/// Change configuration of selected user frame number
FUNCTION_BLOCK WriteFrameDataFB EXTENDS RobotLibraryBaseFB
// ------------------------------------------------------------------------- 
//  SRCI Robot Library                                                
// ------------------------------------------------------------------------- 
//                                                                           
//  Object:      WriteFrameDataFB                                       
//  Author:      Thorsten Brach                                                
//  Date:        2024-06-01
//
//  Description:                                              
//   
//                                                                           
//  Copyright: 
//    (C) 2024 Thorsten Brach. All rights reserved                                                                         
//                                                                           
//  Disclaimer:                                                                           
//    This project is provided without any guarantee and can be used for   
//    private and commercial purposes. Any commercial use is at the user’s 
//    own risk and responsibility.
//
// -------------------------------------------------------------------------
VAR_INPUT 
  /// Start of the command at the rising edge
  Execute            : BOOL;
  /// Processing Mode
  ProcessingMode     : ProcessingMode;
  /// Frame index M
  /// • 0: WCS (default) O
  /// • 1..254: UCS (User frames)
  FrameNo            : USINT;
  /// Frame data (see chapter 5.5.6.2)
  FrameData          : FrameData;
  /// Defines the target sequence in which the command will be executed
  SequenceFlag       : SequenceFlag;
END_VAR
VAR_OUTPUT
  /// The command has been completed successfully
  Done               : BOOL;
  /// FB is being processed
  Busy               : BOOL;
  /// Command is transferred and confirmed by the RC
  CommandBuffered    : BOOL;
  /// The command was aborted by another command
  CommandAborted     : BOOL;
  /// TRUE, while command is interrupted during execution and can be continued.
  CommandInterrupted : BOOL;
END_VAR

                  
                

METHOD PROTECTED OnCall
VAR_IN_OUT
  /// Robot assignment of function
  AxesGroup         : AxesGroup; 
END_VAR
                        
                      
END_METHOD
END_FUNCTION_BLOCK

/// Write integer values on RC
FUNCTION_BLOCK WriteIntegersFB EXTENDS RobotLibraryBaseFB
// ------------------------------------------------------------------------- 
//  SRCI Robot Library                                                
// ------------------------------------------------------------------------- 
//                                                                           
//  Object:      WriteIntegersFB                                       
//  Author:      Thorsten Brach                                                
//  Date:        2024-06-01
//
//  Description:                                              
//   
//                                                                           
//  Copyright: 
//    (C) 2024 Thorsten Brach. All rights reserved                                                                         
//                                                                           
//  Disclaimer:                                                                           
//    This project is provided without any guarantee and can be used for   
//    private and commercial purposes. Any commercial use is at the user’s 
//    own risk and responsibility.
//
// -------------------------------------------------------------------------
VAR_INPUT
  /// Start of the command at the rising edge
  Execute            : BOOL;
  /// Processing Mode
  ProcessingMode     : ProcessingMode;
  /// Specifies the desired target values that shall be written
  Index              : ARRAY[0..6] OF USINT; 
  /// Array value of integers
  Values             : ARRAY[0..6] OF INT;
  /// Set TRUE to prioritize the execution of this command in the defined target sequence.
  HighPriority       : BOOL;
  /// Defines the target sequence in which the command will be executed
  SequenceFlag       : SequenceFlag;
  /// ID of associated trigger function:
  /// •  0: No Trigger (default)  No trigger related behavior
  /// • >0: Trigger - Start executing when the trigger function with the identical EmitterID is triggered.
  /// Always positive.
  /// For more information, see chapter 5.5.12 Triggers
  ListenerID         : SINT;
END_VAR
VAR_OUTPUT
  /// The command has been completed successfully
  Done               : BOOL;
  /// FB is being processed
  Busy               : BOOL;
  /// Command is transferred and confirmed by the RC
  CommandBuffered    : BOOL;
  /// The command was aborted by another command.
  CommandAborted     : BOOL;
  /// TRUE, while command is interrupted during execution and can be continued
  CommandInterrupted : BOOL;
  /// Receiving of input parameter values has been acknowledged by RC
  ParameterAccepted  : BOOL;
  /// Unique system-generated ID of the "Action" when the function is triggered.
  /// • >0: The "Action" is started by the trigger function with identical FollowID.
  /// • <0: The "Action" is stopped by the trigger function with identical FollowID.
  /// For more information see chapter 5.5.12.4.
  OriginID           : USINT;
  /// Relates to ListenerID >0 
  /// Number of successful trigger -based command invocations
  /// For more information refer to chapter 5.5.12.4.
  InvocationCounter  : USINT;
END_VAR

                  
                

METHOD PROTECTED OnCall
VAR_IN_OUT
  /// Robot assignment of function
  AxesGroup         : AxesGroup; 
END_VAR
                        
                      
END_METHOD
END_FUNCTION_BLOCK

/// Change configuration of selected payload number
FUNCTION_BLOCK WriteLoadDataFB EXTENDS RobotLibraryBaseFB
// ------------------------------------------------------------------------- 
//  SRCI Robot Library                                                
// ------------------------------------------------------------------------- 
//                                                                           
//  Object:      WriteLoadDataFB                                       
//  Author:      Thorsten Brach                                                
//  Date:        2024-06-01
//
//  Description:                                              
//   
//                                                                           
//  Copyright: 
//    (C) 2024 Thorsten Brach. All rights reserved                                                                         
//                                                                           
//  Disclaimer:                                                                           
//    This project is provided without any guarantee and can be used for   
//    private and commercial purposes. Any commercial use is at the user’s 
//    own risk and responsibility.
//
// -------------------------------------------------------------------------
VAR_INPUT
  /// Start of the command at the rising edge
  Execute            : BOOL;
  /// Processing Mode
  ProcessingMode     : ProcessingMode;
  /// Load index
  /// •      0: (default) - Not possible to write
  /// • 1..254: Load data
  LoadNo             : USINT;
  /// Load data (see chapter 5.5.6.4)
  LoadData           : LoadData;
  /// Defines the target sequence in which the command will be executed
  SequenceFlag       : SequenceFlag;
END_VAR
VAR_OUTPUT
  /// The command has been completed successfully
  Done               : BOOL;
  /// FB is being processed
  Busy               : BOOL;
  /// Command is transferred and confirmed by the RC
  CommandBuffered    : BOOL;
  /// The command was aborted by another command
  CommandAborted     : BOOL;
  /// TRUE, while command is interrupted during execution and can be continued.
  CommandInterrupted : BOOL;
END_VAR

                  
                

METHOD PROTECTED OnCall
VAR_IN_OUT
  /// Robot assignment of function
  AxesGroup         : AxesGroup; 
END_VAR
                        
                      
END_METHOD
END_FUNCTION_BLOCK

/// Write real values on RC
FUNCTION_BLOCK WriteRealsFB EXTENDS RobotLibraryBaseFB
// ------------------------------------------------------------------------- 
//  SRCI Robot Library                                                
// ------------------------------------------------------------------------- 
//                                                                           
//  Object:      WriteRealsFB                                       
//  Author:      Thorsten Brach                                                
//  Date:        2024-06-01
//
//  Description:                                              
//   
//                                                                           
//  Copyright: 
//    (C) 2024 Thorsten Brach. All rights reserved                                                                         
//                                                                           
//  Disclaimer:                                                                           
//    This project is provided without any guarantee and can be used for   
//    private and commercial purposes. Any commercial use is at the user’s 
//    own risk and responsibility.
//
// -------------------------------------------------------------------------
VAR_INPUT
  /// Start of the command at the rising edge
  Execute            : BOOL;
  /// Processing Mode
  ProcessingMode     : ProcessingMode;
  /// Specifies the desired target values that shall be written
  Index              : ARRAY[0..6] OF USINT; 
  /// Array value of reas
  Values             : ARRAY[0..6] OF REAL;
  /// Set TRUE to prioritize the execution of this command in the defined target sequence.
  HighPriority       : BOOL;
  /// Defines the target sequence in which the command will be executed
  SequenceFlag       : SequenceFlag;
  /// ID of associated trigger function:
  /// •  0: No Trigger (default)  No trigger related behavior
  /// • >0: Trigger - Start executing when the trigger function with the identical EmitterID is triggered.
  /// Always positive.
  /// For more information, see chapter 5.5.12 Triggers
  ListenerID         : SINT;
END_VAR
VAR_OUTPUT
  /// The command has been completed successfully
  Done               : BOOL;
  /// FB is being processed
  Busy               : BOOL;
  /// Command is transferred and confirmed by the RC
  CommandBuffered    : BOOL;
  /// The command was aborted by another command.
  CommandAborted     : BOOL;
  /// TRUE, while command is interrupted during execution and can be continued
  CommandInterrupted : BOOL;
  /// Receiving of input parameter values has been acknowledged by RC
  ParameterAccepted  : BOOL;
  /// Unique system-generated ID of the "Action" when the function is triggered.
  /// • >0: The "Action" is started by the trigger function with identical FollowID.
  /// • <0: The "Action" is stopped by the trigger function with identical FollowID.
  /// For more information see chapter 5.5.12.4.
  OriginID           : USINT;
  /// Relates to ListenerID >0 
  /// Number of successful trigger -based command invocations
  /// For more information refer to chapter 5.5.12.4.
  InvocationCounter  : USINT;
END_VAR

                  
                

METHOD PROTECTED OnCall
VAR_IN_OUT
  /// Robot assignment of function
  AxesGroup         : AxesGroup; 
END_VAR
                        
                      
END_METHOD
END_FUNCTION_BLOCK

/// Write default values of dynamic parameters used by move commands
FUNCTION_BLOCK WriteRobotDefaultDynamicsFB EXTENDS RobotLibraryBaseFB
// ------------------------------------------------------------------------- 
//  SRCI Robot Library                                                
// ------------------------------------------------------------------------- 
//                                                                           
//  Object:      WriteRobotDefaultDynamicsFB                                       
//  Author:      Thorsten Brach                                                
//  Date:        2024-06-01
//
//  Description:                                              
//   
//                                                                           
//  Copyright: 
//    (C) 2024 Thorsten Brach. All rights reserved                                                                         
//                                                                           
//  Disclaimer:                                                                           
//    This project is provided without any guarantee and can be used for   
//    private and commercial purposes. Any commercial use is at the user’s 
//    own risk and responsibility.
//
// -------------------------------------------------------------------------
VAR_INPUT
  /// Start of the command at the rising edge
  Execute                : BOOL;
  /// Processing Mode
  ProcessingMode         : ProcessingMode;
  /// Default dynamics values according to Table 6-141.
  DynamicValues          : DefaultDynamics;
END_VAR
VAR_OUTPUT
  /// The command has been completed successfully
  Done                   : BOOL;
  /// FB is being processed
  Busy                   : BOOL;
  /// Command is transferred and confirmed by the RC
  CommandBuffered        : BOOL;
  /// The command was aborted by another command
  CommandAborted         : BOOL;
  /// TRUE, while command is interrupted during execution and can be continued.
  CommandInterrupted     : BOOL;
  /// Commanded dynamics values according to Table 6-141.
  DefaultDynamicValues   : DefaultDynamics;
END_VAR

                  
                

METHOD PROTECTED OnCall
VAR_IN_OUT
  /// Robot assignment of function
  AxesGroup         : AxesGroup; 
END_VAR
                        
                      
END_METHOD
END_FUNCTION_BLOCK

/// Write reference values of robot dynamics for path movement
FUNCTION_BLOCK WriteRobotReferenceDynamicsFB EXTENDS RobotLibraryBaseFB
// ------------------------------------------------------------------------- 
//  SRCI Robot Library                                                
// ------------------------------------------------------------------------- 
//                                                                           
//  Object:      WriteRobotReferenceDynamicsFB                                       
//  Author:      Thorsten Brach                                                
//  Date:        2024-06-01
//
//  Description:                                              
//   
//                                                                           
//  Copyright: 
//    (C) 2024 Thorsten Brach. All rights reserved                                                                         
//                                                                           
//  Disclaimer:                                                                           
//    This project is provided without any guarantee and can be used for   
//    private and commercial purposes. Any commercial use is at the user’s 
//    own risk and responsibility.
//
// -------------------------------------------------------------------------
VAR_INPUT
  /// Start of the command at the rising edge
  Execute                : BOOL;
  /// Processing Mode
  ProcessingMode         : ProcessingMode;
  /// Reference dynamics values according TO Table 6-134.
  DynamicValues          : ReferenceDynamics;
END_VAR
VAR_OUTPUT
  /// The command has been completed successfully
  Done                   : BOOL;
  /// FB is being processed
  Busy                   : BOOL;
  /// Command is transferred and confirmed by the RC
  CommandBuffered        : BOOL;
  /// The command was aborted by another command
  CommandAborted         : BOOL;
  /// TRUE, while command is interrupted during execution and can be continued.
  CommandInterrupted     : BOOL;
  /// Commanded reference dynamics values according to Table 6-134
  ReferenceDynamicValues : ReferenceDynamics;
END_VAR

                  
                

METHOD PROTECTED OnCall
VAR_IN_OUT
  /// Robot assignment of function
  AxesGroup         : AxesGroup; 
END_VAR
                        
                      
END_METHOD
END_FUNCTION_BLOCK

/// Change robot limits of robot axes (degree)
FUNCTION_BLOCK WriteRobotSWLimitsFB EXTENDS RobotLibraryBaseFB
// ------------------------------------------------------------------------- 
//  SRCI Robot Library                                                
// ------------------------------------------------------------------------- 
//                                                                           
//  Object:      WriteRobotSWLimitsFB                                       
//  Author:      Thorsten Brach                                                
//  Date:        2024-06-01
//
//  Description:                                              
//   
//                                                                           
//  Copyright: 
//    (C) 2024 Thorsten Brach. All rights reserved                                                                         
//                                                                           
//  Disclaimer:                                                                           
//    This project is provided without any guarantee and can be used for   
//    private and commercial purposes. Any commercial use is at the user’s 
//    own risk and responsibility.
//
// -------------------------------------------------------------------------
VAR_INPUT
  /// Start of the command at the rising edge
  Execute                : BOOL;
  /// Limits for joints and external axes according to Table 6-180.
  LimitValues            : SWLimits;
  /// Reset limits to RC specific factory settings
  ResetToFactoryDefaults : BOOL;;
END_VAR
VAR_OUTPUT
  /// The command has been completed successfully
  Done                   : BOOL;
  /// FB is being processed
  Busy                   : BOOL;
  /// Command is transferred and confirmed by the RC
  CommandBuffered        : BOOL;
  /// TRUE, when Software limits were overwritten but not activated on RC until a restart of the RC
  RestartRequested       : BOOL;
END_VAR

                  
                

METHOD PROTECTED OnCall
VAR_IN_OUT
  /// Robot assignment of function
  AxesGroup         : AxesGroup; 
END_VAR
                        
                      
END_METHOD
END_FUNCTION_BLOCK

/// Write specific parameter of the robot
FUNCTION_BLOCK WriteSystemVariableFB EXTENDS RobotLibraryBaseFB
// ------------------------------------------------------------------------- 
//  SRCI Robot Library                                                
// ------------------------------------------------------------------------- 
//                                                                           
//  Object:      WriteSystemVariableFB                                       
//  Author:      Thorsten Brach                                                
//  Date:        2024-06-01
//
//  Description:                                              
//   
//                                                                           
//  Copyright: 
//    (C) 2024 Thorsten Brach. All rights reserved                                                                         
//                                                                           
//  Disclaimer:                                                                           
//    This project is provided without any guarantee and can be used for   
//    private and commercial purposes. Any commercial use is at the user’s 
//    own risk and responsibility.
//
// -------------------------------------------------------------------------
VAR_INPUT
  /// Start of the command at the rising edge
  Execute            : BOOL;
  /// Processing Mode
  ProcessingMode     : ProcessingMode;
  /// Defines the parameter list which should be used:
  /// • FALSE: Standardized parameter list (default):
  ///          -  Read parameters on the RC based on a standardized parameter list
  /// • TRUE: Manufacturer specific parameter list:
  ///        -  Read parameters on the RC based on robot manufacturers-specific parameter lists
  RCParameter        : BOOL;
  /// Requested parameter ID in selected parameter list.
  /// •          0: undefined (default)
  /// • 1..65 535: Parameter ID
  ParameterID        : ARRAY[0..7] OF UINT;
  /// ID of the requested sub parameter in selected parameter list.
  /// • 0: ID 0 (default) (relates only to parameters without sub parameters)
  /// • 1..255: Indices 1 to 255 (relates only to parameters with sub parameters)
  SubParameterID     : ARRAY[0..7] OF USINT;  
  /// Parameter data type as specified in Table 6-621.
  DataType           : ARRAY[0..7] OF USINT;
  /// Parameter data addressed by input values of ParameterID[0] and SubParameterID[0]
  Data_0             : ARRAY[0..3] OF BYTE;
  /// Parameter data addressed by input values of ParameterID[1] and SubParameterID[1]
  Data_1             : ARRAY[0..3] OF BYTE;
  /// Parameter data addressed by input values of ParameterID[2] and SubParameterID[2]
  Data_2             : ARRAY[0..3] OF BYTE;
  /// Parameter data addressed by input values of ParameterID[3] and SubParameterID[3]
  Data_3             : ARRAY[0..3] OF BYTE;
  /// Parameter data addressed by input values of ParameterID[4] and SubParameterID[4]
  Data_4             : ARRAY[0..3] OF BYTE;
  /// Parameter data addressed by input values of ParameterID[5] and SubParameterID[5]
  Data_5             : ARRAY[0..3] OF BYTE;
  /// Parameter data addressed by input values of ParameterID[6] and SubParameterID[6]
  Data_6             : ARRAY[0..3] OF BYTE;
  /// Parameter data addressed by input values of ParameterID[7] and SubParameterID[7]
  Data_7             : ARRAY[0..3] OF BYTE;
  /// Defines the target sequence in which the command will be executed
  SequenceFlag       : SequenceFlag;
  /// ID of associated trigger function:
  /// •  0: No Trigger (default)  No trigger related behavior
  /// • >0: Trigger - Start executing when the trigger function with the identical EmitterID is triggered.
  /// Always positive.
  /// For more information, see chapter 5.5.12 Triggers
  ListenerID         : SINT;
END_VAR
VAR_OUTPUT
  /// The command has been completed successfully
  Done               : BOOL;
  /// FB is being processed
  Busy               : BOOL;
  /// Command is transferred and confirmed by the RC
  CommandBuffered    : BOOL;
  /// The command was aborted by another command.
  CommandAborted     : BOOL;
  /// TRUE, while command is interrupted during execution and can be continued
  CommandInterrupted : BOOL;
  /// TRUE, when parameters were overwritten but not activated on RC until a restart of the RC
  RestartRequested   : BOOL;
  /// Unique system-generated ID of the "Action" when the function is triggered.
  /// • >0: The "Action" is started by the trigger function with identical FollowID.
  /// • <0: The "Action" is stopped by the trigger function with identical FollowID.
  /// For more information see chapter 5.5.12.4 EmitterID, ListenerID, FollowID and OriginID
  OriginID           : INT;
  /// Relates to ListenerID >0
  /// Number of successful trigger -based command invocations
  /// For more information refer to chapter 5.5.12.4.
  InvocationCounter  : USINT;
END_VAR

                  
                

METHOD PROTECTED OnCall
VAR_IN_OUT
  /// Robot assignment of function
  AxesGroup         : AxesGroup; 
END_VAR
                        
                      
END_METHOD
END_FUNCTION_BLOCK

/// Change configuration of selected tool number
FUNCTION_BLOCK WriteToolDataFB EXTENDS RobotLibraryBaseFB
// ------------------------------------------------------------------------- 
//  SRCI Robot Library                                                
// ------------------------------------------------------------------------- 
//                                                                           
//  Object:      WriteToolDataFB                                       
//  Author:      Thorsten Brach                                                
//  Date:        2024-06-01
//
//  Description:                                              
//   
//                                                                           
//  Copyright: 
//    (C) 2024 Thorsten Brach. All rights reserved                                                                         
//                                                                           
//  Disclaimer:                                                                           
//    This project is provided without any guarantee and can be used for   
//    private and commercial purposes. Any commercial use is at the user’s 
//    own risk and responsibility.
//
// -------------------------------------------------------------------------
VAR_INPUT
  /// Start of the command at the rising edge
  Execute            : BOOL;
  /// Processing Mode
  ProcessingMode     : ProcessingMode;
  /// Tool index
  /// •      0: Flange (default) Not possible to change
  /// • 1..254: Tool Frame
  ToolNo            : USINT;
  /// Tool data (see chapter 5.5.6.3)
  ToolData          : ToolData;
  /// Defines the target sequence in which the command will be executed
  SequenceFlag       : SequenceFlag;
END_VAR
VAR_OUTPUT
  /// The command has been completed successfully
  Done               : BOOL;
  /// FB is being processed
  Busy               : BOOL;
  /// Command is transferred and confirmed by the RC
  CommandBuffered    : BOOL;
  /// The command was aborted by another command
  CommandAborted     : BOOL;
  /// TRUE, while command is interrupted during execution and can be continued.
  CommandInterrupted : BOOL;
END_VAR

                  
                

METHOD PROTECTED OnCall
VAR_IN_OUT
  /// Robot assignment of function
  AxesGroup         : AxesGroup; 
END_VAR
                        
                      
END_METHOD
END_FUNCTION_BLOCK

/// Define work area
FUNCTION_BLOCK WriteWorkAreaFB EXTENDS RobotLibraryBaseFB
// ------------------------------------------------------------------------- 
//  SRCI Robot Library                                                
// ------------------------------------------------------------------------- 
//                                                                           
//  Object:      WriteWorkAreaFB                                       
//  Author:      Thorsten Brach                                                
//  Date:        2024-06-01
//
//  Description:                                              
//   
//                                                                           
//  Copyright: 
//    (C) 2024 Thorsten Brach. All rights reserved                                                                         
//                                                                           
//  Disclaimer:                                                                           
//    This project is provided without any guarantee and can be used for   
//    private and commercial purposes. Any commercial use is at the user’s 
//    own risk and responsibility.
//
// -------------------------------------------------------------------------
VAR_INPUT
  /// Start of the command at the rising edge
  Execute            : BOOL;
  /// Processing Mode
  ProcessingMode     : ProcessingMode;
  /// Index of the robot work area
  /// • 0 (default)..254
  WorkAreaNo         : USINT;
  /// Data specific to the work area requested by Index.
  WorkAreaData       : RobotWorkArea;
END_VAR
VAR_OUTPUT
  /// The command has been completed successfully
  Done               : BOOL;
  /// FB is being processed
  Busy               : BOOL;
  /// Command is transferred and confirmed by the RC
  CommandBuffered    : BOOL;
END_VAR

                  
                

METHOD PROTECTED OnCall
VAR_IN_OUT
  /// Robot assignment of function
  AxesGroup         : AxesGroup; 
END_VAR
                        
                      
END_METHOD
END_FUNCTION_BLOCK

FUNCTION_BLOCK ActiveCommandRegisterFB
// ------------------------------------------------------------------------- 
//  SRCI Robot Library                                                
// ------------------------------------------------------------------------- 
//                                                                           
//  Object:      ActiveCommandRegisterFB                                       
//  Author:      Thorsten Brach                                                
//  Date:        2024-06-01
//
//  Description:                                              
//   
//                                                                           
//  Copyright: 
//    (C) 2024 Thorsten Brach. All rights reserved                                                                         
//                                                                           
//  Disclaimer:                                                                           
//    This project is provided without any guarantee and can be used for   
//    private and commercial purposes. Any commercial use is at the user’s 
//    own risk and responsibility.
//
// -------------------------------------------------------------------------
VAR_INPUT
  /// Active Command Register
  Register            : ARRAY [1..RobotLibraryParameter.ACTIVE_CMD_REGISTER_ENTRIES_MAX] OF AxesGroupAcyclicAcrEntry;
END_VAR

VAR_OUTPUT
  /// Size of the register 
  Size                : UINT := DINT_TO_UINT(RobotLibraryParameter.ACTIVE_CMD_REGISTER_ENTRIES_MAX);
  /// Execution Order List 
  ExecutionOrderList  : AxesGroupAcyclicExecutionOrderList;
END_VAR

VAR
  /// last used unique ID 
  LastUniqueID        : UDINT;
END_VAR

                  OnCall();


                

METHOD INTERNAL AddCmd : UDINT
VAR_INPUT
  /// Reference to the corresponding command-FB to enable a callback mechanism
  rCommandFB   : REFERENCE TO RobotLibraryBaseFB;
END_VAR

VAR
  /// internal index for loops
 _idx : DINT;
END_VAR
                        FOR _idx := 1 TO RobotLibraryParameter.ACTIVE_CMD_REGISTER_ENTRIES_MAX
DO
  IF ( Register[_idx].State = ActiveCommandRegisterState.IS_FREE )
  THEN
    Register[_idx].State                        := ActiveCommandRegisterState.IS_PROCESSING;
    Register[_idx].UniqueID                     := CreateUniqueID();
    Register[_idx].rCommandFB                   := rCommandFB;

    // check reference to command FB
    IF (__ISVALIDREF(Register[_idx].rCommandFB))
    THEN
      Register[_idx].Command[1].Payload    := rCommandFB.CommandData.Payload;
      Register[_idx].Command[1].PayloadLen := rCommandFB.CommandData.PayloadLen;
      Register[_idx].Command[1].PayLoadPtr := 0;
      Register[_idx].Command[1].State      := BufferStateCmd.CREATED;
		END_IF
  
    // return Unique ID
    AddCmd := Register[_idx].UniqueID;
    EXIT;
	END_IF
END_FOR
                      
END_METHOD

METHOD INTERNAL CreateUniqueID : UDINT
VAR_INPUT
END_VAR
                        // inc last unique ID 
LastUniqueID := LastUniqueID + 1;
// return unique ID
CreateUniqueID := LastUniqueID;
                      
END_METHOD

METHOD INTERNAL OnCall
                        
                      
END_METHOD

METHOD OnlineChange : DINT
VAR_INPUT
  /// unique ID 
  UniqueID     : UDINT;
  /// Reference to the corresponding command-FB to enable a callback mechanism
  rCommandFB   : REFERENCE TO RobotLibraryBaseFB;
END_VAR

VAR
  /// internal index for loops
 _idx : DINT;
END_VAR
                        OnlineChange := -1;

// Check command FB reference is valid ?
IF ( NOT __ISVALIDREF(rCommandFB))
THEN
  RETURN;
END_IF

FOR _idx := 1 TO RobotLibraryParameter.ACTIVE_CMD_REGISTER_ENTRIES_MAX
DO
  // check unique ID found ?
  IF ( Register[_idx].UniqueID = UniqueID ) 
  THEN  
    // update reference to command FB
    Register[_idx].rCommandFB := rCommandFB;
    // Return result OK
    OnlineChange := RobotLibraryConstants.OK;
    EXIT;
  END_IF
END_FOR
                      
END_METHOD

METHOD RemoveCmd
VAR_INPUT
 /// unique ID
 UniqueID : UDINT;  
END_VAR

VAR
  /// internal index
 _idx : DINT;
END_VAR
                        FOR _idx := 1 TO RobotLibraryParameter.ACTIVE_CMD_REGISTER_ENTRIES_MAX
DO
  // check unique ID found and not yet sended ?
  IF (( Register[_idx].UniqueID         = UniqueID               ) AND
      ( Register[_idx].Command[1].State < BufferStateCmd.SENDING ))       
  THEN  
    // delete register entry
    MemSet(ADR(Register[_idx]), 0 , SIZEOF(Register[_idx]));
    EXIT;
  END_IF
END_FOR
                      
END_METHOD

METHOD SortList : ARRAY [1..RobotLibraryParameter.ACTIVE_CMD_REGISTER_ENTRIES_MAX] OF UINT;
VAR_INPUT
  List : ARRAY [1..RobotLibraryParameter.ACTIVE_CMD_REGISTER_ENTRIES_MAX] OF UINT;
END_VAR

VAR
  i   : DINT;
  j   : DINT;
  tmp : UINT;
END_VAR
                        // Bubble Sort 
FOR i := 1 TO RobotLibraryParameter.ACTIVE_CMD_REGISTER_ENTRIES_MAX
DO
  FOR j := 1 TO RobotLibraryParameter.ACTIVE_CMD_REGISTER_ENTRIES_MAX - 1
  DO
    IF ( List[j] > List[j+1])
    THEN
       Tmp := List[j];         
       List[j]   := List[j+1];
       List[j+1] := Tmp;
    END_IF
  END_FOR 
END_FOR

// return sorted list
SortList := List;
                      
END_METHOD

METHOD UpdateExecutionOrderList
VAR
  _idxReg  : DINT;
  _idxList : DINT := 1;
END_VAR
                        FOR _idxReg := 1 TO RobotLibraryParameter.ACTIVE_CMD_REGISTER_ENTRIES_MAX
DO
  IF (( Register[_idxReg].State              = ActiveCommandRegisterState.IS_PROCESSING ) AND
      ( Register[_idxReg].Response[1].State  =             BufferStateRsp.EMPTY         ))     
  THEN
    ;
  END_IF
END_FOR
                      
END_METHOD
END_FUNCTION_BLOCK

{attribute 'pack_mode' := '1'} 
FUNCTION_BLOCK RecvData
// ------------------------------------------------------------------------- 
//  SRCI Robot Library                                                
// ------------------------------------------------------------------------- 
//                                                                           
//  Object:      RecvData                                       
//  Author:      Thorsten Brach                                                
//  Date:        2024-06-01
//
//  Description:                                              
//   
//                                                                           
//  Copyright: 
//    (C) 2024 Thorsten Brach. All rights reserved                                                                         
//                                                                           
//  Disclaimer:                                                                           
//    This project is provided without any guarantee and can be used for   
//    private and commercial purposes. Any commercial use is at the user’s 
//    own risk and responsibility.
//
// -------------------------------------------------------------------------
VAR_INPUT
  /// Payload
  Payload    : ARRAY [0..RobotLibraryParameter.TELEGRAM_PAYLOAD_MAX] OF BYTE;
  /// Payload length
  PayloadLen : UDINT;
  /// Payload pointer
  PayloadPtr : DINT;
END_VAR

                  
                

/// returns a ArmConfigParameter from the payload buffer from the current payload pointer address and increase the payload pointer afterwards
METHOD GetArmConfig : ArmConfigParameter
VAR
  /// temporary byte
 _tmpByte : BYTE;
END_VAR
                        // get 1st Byte
_tmpByte := GetByte();

GetArmConfig.Shoulder.0 := _tmpByte.0;
GetArmConfig.Elbow.0    := _tmpByte.1;
GetArmConfig.Wrist.0    := _tmpByte.2;

// get 2nd byte to inc the PayloadPointer
_tmpByte := GetByte();
                      
END_METHOD

/// returns a BOOL from the payload buffer from the current payload pointer address and increase the payload pointer afterwards
METHOD GetBool : BOOL
                        // copy data
GetBool := Payload[PayloadPtr].0;
// inc payload pointer 
PayloadPtr := PayloadPtr + SIZEOF(BYTE);
                      
END_METHOD

/// returns a BYTE from the payload buffer from the current payload pointer address and increase the payload pointer afterwards
METHOD GetByte : BYTE
                        // copy data
GetByte := Payload[PayloadPtr];
// inc payload pointer 
PayloadPtr := PayloadPtr + SIZEOF(BYTE);
                      
END_METHOD

/// returns a DWORD from the payload buffer from the current payload pointer address and increase the payload pointer afterwards
METHOD GetDword : DWORD
                        // copy data
MemCpy(ADR(GetDword), ADR(Payload[PayloadPtr]), SIZEOF(DWORD));
// inc payload pointer 
PayloadPtr := PayloadPtr + SIZEOF(DWORD);
                      
END_METHOD

/// returns the 1st halfe BYTE from the payload buffer from the current payload pointer address and increase the payload pointer afterwards
METHOD GetHalfeByte1 : BYTE
VAR_INPUT
  /// Increase payload pointer 
  IncPayloadPtr : BOOL;
END_VAR

VAR
  /// temporary byte
 _tmpByte : BYTE;
END_VAR
                        // copy data
_tmpByte := Payload[PayloadPtr];

GetHalfeByte1.0 := _tmpByte.0;
GetHalfeByte1.1 := _tmpByte.1;
GetHalfeByte1.2 := _tmpByte.2;
GetHalfeByte1.3 := _tmpByte.3;


IF (IncPayloadPtr)
THEN  
  // inc payload pointer
  PayloadPtr := PayloadPtr + SIZEOF(BYTE);
END_IF

                      
END_METHOD

/// returns the 1st halfe BYTE from the payload buffer from the current payload pointer address and increase the payload pointer afterwards
METHOD GetHalfeByte2 : BYTE
VAR_INPUT
  /// Increase payload pointer 
  IncPayloadPtr : BOOL;
END_VAR

VAR
  /// temporary byte
 _tmpByte : BYTE;
END_VAR
                        // copy data
_tmpByte := Payload[PayloadPtr];

GetHalfeByte2.0 := _tmpByte.4;
GetHalfeByte2.1 := _tmpByte.5;
GetHalfeByte2.2 := _tmpByte.6;
GetHalfeByte2.3 := _tmpByte.7;

IF (IncPayloadPtr)
THEN  
  // inc payload pointer
  PayloadPtr := PayloadPtr + SIZEOF(BYTE);
END_IF

                      
END_METHOD

/// returns a INT from the payload buffer from the current payload pointer address and increase the payload pointer afterwards
METHOD GetInt : INT
                        // copy data
MemCpy(ADR(GetInt), ADR(Payload[PayloadPtr]), SIZEOF(INT));
// swap byte order
GetInt := SwapInt(GetInt);
// inc payload pointer   
PayloadPtr := PayloadPtr + SIZEOF(INT);
                      
END_METHOD

/// returns a REAL from the payload buffer from the current payload pointer address and increase the payload pointer afterwards
METHOD GetReal : REAL
                        // copy data
MemCpy(ADR(GetReal), ADR(Payload[PayloadPtr]), SIZEOF(REAL));
// swap byte order
GetReal := SwapReal(GetReal);
// inc payload pointer   
PayloadPtr := PayloadPtr + SIZEOF(Real);
                      
END_METHOD

/// returns a SINT from the payload buffer from the current payload pointer address and increase the payload pointer afterwards
METHOD GetSint : SINT
                        // copy data
MemCpy(ADR(GetSint), ADR(Payload[PayloadPtr]), SIZEOF(SINT));
// inc payload pointer 
PayloadPtr := PayloadPtr + SIZEOF(SINT);
                      
END_METHOD

/// returns a TurnNumber from the payload buffer from the current payload pointer address and increase the payload pointer afterwards
METHOD GetTurnNumbers : TurnNumber
                        GetTurnNumbers.J1Turns := BYTE_TO_SINT(GetHalfeByte1(FALSE));
GetTurnNumbers.J2Turns := BYTE_TO_SINT(GetHalfeByte2(TRUE));

GetTurnNumbers.J3Turns := BYTE_TO_SINT(GetHalfeByte1(FALSE));
GetTurnNumbers.J4Turns := BYTE_TO_SINT(GetHalfeByte2(TRUE));

GetTurnNumbers.J5Turns := BYTE_TO_SINT(GetHalfeByte1(FALSE));
GetTurnNumbers.J6Turns := BYTE_TO_SINT(GetHalfeByte2(TRUE));

GetTurnNumbers.E1Turns := BYTE_TO_SINT(GetByte());
                      
END_METHOD

/// returns a UINT from the payload buffer from the current payload pointer address and increase the payload pointer afterwards
METHOD GetUint : UINT
                        // copy data
MemCpy(ADR(GetUint), ADR(Payload[PayloadPtr]), SIZEOF(UINT));
// swap byte order
GetUint := SwapUint(GetUint);
// inc payload pointer   
PayloadPtr := PayloadPtr + SIZEOF(UINT);
                      
END_METHOD

/// returns a USINT from the payload buffer from the current payload pointer address and increase the payload pointer afterwards
METHOD GetUsint : USINT
                        // copy data
MemCpy(ADR(GetUsint), ADR(Payload[PayloadPtr]), SIZEOF(USINT));
// inc payload pointer 
PayloadPtr := PayloadPtr + SIZEOF(USINT);
                      
END_METHOD

/// returns a WORD from the payload buffer from the current payload pointer address and increase the payload pointer afterwards
METHOD GetWord : WORD
                        // copy data
MemCpy(ADR(GetWord), ADR(Payload[PayloadPtr]), SIZEOF(WORD));
// swap byte order
GetWord := SwapWord(GetWord);
// inc payload pointer   
PayloadPtr := PayloadPtr + SIZEOF(WORD);
                      
END_METHOD

/// Resets the payload pointer to start address
METHOD ResetPointer
VAR_INPUT
END_VAR
                        // Reset payload pointer
PayloadPtr := 0;
                      
END_METHOD

/// returns a FragmentAction from the payload buffer from the current payload pointer address and increase the payload pointer afterwards
METHOD GetFragmentAction : FragmentAction
VAR
  /// temporary byte
 _tmpByte : BYTE;
END_VAR
                        // copy data
_tmpByte := Payload[PayloadPtr];

GetFragmentAction.Complete := _tmpByte.0;
GetFragmentAction.Reset    := _tmpByte.1;
GetFragmentAction.Clear    := _tmpByte.2;
GetFragmentAction.BIT03    := _tmpByte.3;
GetFragmentAction.BIT04    := _tmpByte.4;
GetFragmentAction.BIT05    := _tmpByte.5;
GetFragmentAction.BIT06    := _tmpByte.6;
GetFragmentAction.BIT07    := _tmpByte.7;

// inc payload pointer   
PayloadPtr := PayloadPtr + SIZEOF(BYTE);
                      
END_METHOD
END_FUNCTION_BLOCK

{attribute 'pack_mode' := '1'} 
FUNCTION_BLOCK SendData
// ------------------------------------------------------------------------- 
//  SRCI Robot Library                                                
// ------------------------------------------------------------------------- 
//                                                                           
//  Object:      SendData                                      
//  Author:      Thorsten Brach                                                
//  Date:        2024-06-01
//
//  Description:                                              
//    
//                                                                           
//  Copyright: 
//    (C) 2024 Thorsten Brach. All rights reserved                                                                         
//                                                                           
//  Disclaimer:                                                                           
//    This project is provided without any guarantee and can be used for   
//    private and commercial purposes. Any commercial use is at the user’s 
//    own risk and responsibility.
//
// -------------------------------------------------------------------------
VAR_INPUT
  /// Payload
  Payload    : ARRAY [0..RobotLibraryParameter.TELEGRAM_PAYLOAD_MAX] OF BYTE;
  /// Payload length
  PayloadLen : UDINT;
  /// Payload pointer
  PayloadPtr : UDINT;
END_VAR

                  
                

/// Adds a BOOL to the payload buffer, increase the payload pointer and returns the payload lenght
METHOD AddBool : UDINT
VAR_INPUT
  /// Value to add
  Value : BOOL;
END_VAR

VAR
  /// temporary byte
 _tmpByte : BYTE := 0;
END_VAR
                        _tmpByte.0 := Value;
// copy data 
MemCpy( ADR(Payload[PayloadPtr]), ADR(_tmpByte), SIZEOF(_tmpByte));
// inc payload pointer 
PayloadPtr := PayloadPtr + SIZEOF(_tmpByte);
// return payload len
AddBool := PayloadLen := PayloadPtr;
                      
END_METHOD

/// Adds a BYTE to the payload buffer, increase the payload pointer and returns the payload lenght
METHOD AddByte : UDINT
VAR_INPUT
  /// Value to add
  Value : BYTE;
END_VAR
                        Value := Value;
// copy data 
MemCpy( ADR(Payload[PayloadPtr]), ADR(Value), SIZEOF(Value));
// inc payload pointer 
PayloadPtr := PayloadPtr + SIZEOF(Value);
// return payload len
AddByte := PayloadLen := PayloadPtr;
                      
END_METHOD

/// Adds a DataBlock to the payload buffer, increase the payload pointer and returns the payload lenght
METHOD AddDataBlock : UDINT
VAR_INPUT
  /// Value to add
  pValue : POINTER TO BYTE;
  /// Size of data block
  Size   : UDINT;
END_VAR
                        IF (pValue = 0) OR (Size = 0 )
THEN
  RETURN;
END_IF

// copy data 
MemCpy( ADR(Payload[PayloadPtr]), pValue, Size);
// inc payload pointer 
PayloadPtr := PayloadPtr + Size;
// return payload len
AddDataBlock := PayloadLen := PayloadPtr;
                      
END_METHOD

/// Adds two halfe BYTE to the payload buffer , increase the payload pointer and returns the payload lenght
METHOD AddHalfBytes : UDINT
VAR_INPUT
  /// Value to add
  Value1 : BYTE;
  /// Value to add
  Value2 : BYTE;
END_VAR

VAR
  /// internal value
 _value : BYTE;
END_VAR
                        _value := CombineHalfBytes(Value1,Value2);
// copy data 
MemCpy( ADR(Payload[PayloadPtr]), ADR(_value), SIZEOF(_value));
// inc payload pointer 
PayloadPtr := PayloadPtr + SIZEOF(_value);
// return payload len
AddHalfBytes := PayloadLen := PayloadPtr;
                      
END_METHOD

/// Adds a REAL to the payload buffer , increase the payload pointer and returns the payload lenght
METHOD AddReal : UDINT
VAR_INPUT
  /// Value to add
  Value : REAL;
END_VAR
                        // swap byte order
Value := SwapReal(Value);
// copy data 
MemCpy( ADR(Payload[PayloadPtr]), ADR(Value), SIZEOF(Value));
// inc data index 
PayloadPtr := PayloadPtr + SIZEOF(Value);
// return payload len
AddReal := PayloadLen := PayloadPtr;
                      
END_METHOD

/// Adds a SINT to the payload buffer, increase the payload pointer and returns the payload lenght
METHOD AddSint : UDINT
VAR_INPUT
  /// Value to add
  Value : SINT;
END_VAR
                        Value := Value;
// copy data 
MemCpy( ADR(Payload[PayloadPtr]), ADR(Value), SIZEOF(Value));
// inc payload pointer 
PayloadPtr := PayloadPtr + SIZEOF(Value);
// return payload len
AddSint := PayloadLen := PayloadPtr;
                      
END_METHOD

/// Adds a TIME to the payload buffer , increase the payload pointer and returns the payload lenght
METHOD AddTime : UDINT
VAR_INPUT
  /// Value to add
  Value : TOD;
END_VAR
                        // swap byte order
Value := SwapTime(Value);
// copy data 
MemCpy( ADR(Payload[PayloadPtr]), ADR(Value), SIZEOF(Value));
// inc data index 
PayloadPtr := PayloadPtr + SIZEOF(Value);
// return payload len
AddTime := PayloadLen := PayloadPtr;
                      
END_METHOD

/// Adds a UINT to the payload buffer , increase the payload pointer and returns the payload lenght
METHOD AddUint : UDINT
VAR_INPUT
  /// Value to add
  Value : UINT;
END_VAR
                        // swap byte order
Value := SwapUint(Value);
// copy data 
MemCpy( ADR(Payload[PayloadPtr]), ADR(Value), SIZEOF(Value));
// inc data index 
PayloadPtr := PayloadPtr + SIZEOF(Value);
// return payload len
AddUint := PayloadLen := PayloadPtr;
                      
END_METHOD

/// Adds a USINT to the payload buffer, increase the payload pointer and returns the payload lenght
METHOD AddUsint : UDINT
VAR_INPUT
  /// Value to add
  Value : USINT;
END_VAR
                        Value := Value;
// copy data 
MemCpy( ADR(Payload[PayloadPtr]), ADR(Value), SIZEOF(Value));
// inc payload pointer 
PayloadPtr := PayloadPtr + SIZEOF(Value);
// return payload len
AddUsint := PayloadLen := PayloadPtr;
                      
END_METHOD

/// Resets the payload buffer, the payload pointer and the payload length
METHOD Reset
VAR_INPUT
END_VAR
                        MemSet(ADR(Payload), 0 , SIZEOF(Payload));
PayloadLen := 0;
PayloadPtr := 0;
                      
END_METHOD

/// Adds a ArmConfigParameter to the payload buffer, increase the payload pointer and returns the payload lenght
METHOD AddArmConfig : UDINT
VAR_INPUT
  /// Value to add
  Value : ArmConfigParameter;
END_VAR

VAR
  /// temporary Byte
 _tmpByte : BYTE;
END_VAR
                        Value := Value;

_tmpByte.0 := Value.Shoulder.0;
_tmpByte.1 := Value.Elbow.0;
_tmpByte.2 := Value.Wrist.0;

AddByte(_tmpByte);
AddByte(0);

AddArmConfig := PayloadLen; 

                      
END_METHOD

/// Adds a TurnNumber to the payload buffer, increase the payload pointer and returns the payload lenght
METHOD AddTurnNumber : UDINT
VAR_INPUT
  /// Value to add
  Value : TurnNumber;
END_VAR

VAR
  /// temporary Byte
 _tmpByte : BYTE;
END_VAR
                        Value := Value;

AddHalfBytes( SINT_TO_BYTE(Value.J1Turns) , SINT_TO_BYTE(Value.J2Turns));
AddHalfBytes( SINT_TO_BYTE(Value.J3Turns) , SINT_TO_BYTE(Value.J4Turns));
AddHalfBytes( SINT_TO_BYTE(Value.J5Turns) , SINT_TO_BYTE(Value.J6Turns));
AddByte(SINT_TO_BYTE(Value.E1Turns));

AddTurnNumber := PayloadLen; 

                      
END_METHOD
END_FUNCTION_BLOCK

/// Enable/Disable work areas of RC and check if TCP is inside/outside of active work area
FUNCTION_BLOCK ActivateWorkAreaFB EXTENDS RobotLibraryBaseFB
// ------------------------------------------------------------------------- 
//  SRCI Robot Library                                                
// ------------------------------------------------------------------------- 
//                                                                           
//  Object:      ActivateWorkAreaFB                                       
//  Author:      Thorsten Brach                                                
//  Date:        2024-06-01
//
//  Description:                                              
//   
//                                                                           
//  Copyright: 
//    (C) 2024 Thorsten Brach. All rights reserved                                                                         
//                                                                           
//  Disclaimer:                                                                           
//    This project is provided without any guarantee and can be used for   
//    private and commercial purposes. Any commercial use is at the user’s 
//    own risk and responsibility.
//
// -------------------------------------------------------------------------
VAR_INPUT
  /// Start of the command at the rising edge
  Execute         : BOOL;
  /// Command parameter
  ParCmd          : ActivateWorkAreaParCmd;
END_VAR
VAR_OUTPUT
  /// The command has been completed successfully
  Done            : BOOL;
  /// FB is being processed
  Busy            : BOOL;
  /// Command is transferred and confirmed by the RC
  CommandBuffered : BOOL;
  /// Command parameter
  OutCmd          : ActivateWorkAreaOutCmd;
END_VAR
VAR
  /// internal copy of command parameter 
 _parCmd          : ActivateWorkAreaParCmd;
  /// command data to send
 _command         : ActivateWorkAreaSendData;
  /// response data received
 _response        : ActivateWorkAreaRecvData;    
END_VAR

                  
                

METHOD CheckParameterChanged : BOOL
                        // compare memory 
CheckParameterChanged := ( MemCmp(ADR(ParCmd), ADR(_parCmd), SIZEOF(ParCmd)) = RobotLibraryConstants.OK );

IF ( CheckParameterChanged )
THEN  
  // update internal copy of parameters 
 _parCmd := ParCmd;
  // inc parameter sequence
 _command.ParSeq := _command.ParSeq + 1;
  // update command data  
  CommandData := CreateCommandData(); // ( Access via reference to rCommandFB in ACR )
END_IF
                      
END_METHOD

METHOD CreateCommandData : SendData
                        // Table 6-211: Sent CMD payload (PLC to RC) of "ActivateWorkArea"

// --------------------------
// Header
// --------------------------
// Byte 00 : UINT  - Type HB     
// Byte 01 :       - Type LB    
// Byte 02 : USINT - Reserve | ExecutionMode
// Byte 03 : USINT - ParSeq  | Priority
// --------------------------
// Datablock
// --------------------------
// Byte 04 : USINT - WorkAreaNo
// Byte 05 : BOOL  - ActivateArea
// --------------------------

// set command parameter 
_command.CmdTyp       :=  CmdType.ActivateWorkArea;
_command.ExecMode     :=  ExecutionMode.PARALLEL;
_command.ParSeq       := _command.ParSeq;
_command.Priority     :=  PriorityLevel.NORMAL;
_command.WorkAreaNo   := _parCmd.WorkAreaNo;
_command.ActivateArea := _parCmd.ActivateArea;


// copy command data to header
_cmdHeader := _command;
// call base implementation to copy header to payload buffer
SUPER^.CreateCommandData();

// add command.WorkAreaNo
CreateCommandData.AddUsint(_command.WorkAreaNo);
// add command.ActivateArea
CreateCommandData.AddBool(_command.ActivateArea);

                      
END_METHOD

METHOD PROTECTED OnCall
VAR_IN_OUT
  /// Robot assignment of function
  AxesGroup : AxesGroup; 
END_VAR
                        CASE _stepCmd OF
  
  00:  IF ( Execute ) 
       THEN
         // set busy flag
         Busy := TRUE;
         // Reset command outputs
         MemSet(ADR(OutCmd),0,SIZEOF(OutCmd));         
         // apply command parameter
        _parCmd := ParCmd;
         // init parameter sequence
        _command.ParSeq := 1;
         // set timeout
         SetTimeout(PT := _timeoutCmd, rTimer := _timerCmd);
         // inc step counter
        _stepCmd := _stepCmd + 1; 
	     END_IF
     
  01:  // create command data
       CommandData := CreateCommandData();
       // Add command to active command register
      _uniqueID := AxesGroup.Acyclic.ActiveCommandRegister.AddCmd( rCommandFB := THIS^ );     
       // set timeout
       SetTimeout(PT := _timeoutCmd, rTimer := _timerCmd);
       // inc step counter
      _stepCmd := _stepCmd + 1; 

  02:  // Wait for responce received
       IF ( _responseReceived )
       THEN
         // reset response received flag
        _responseReceived := FALSE;

         CASE  _response.State 
         OF
           CmdMessageState.BUFFERED    : CommandBuffered    := TRUE;
         //CmdMessageState.ACTIVE      : Active             := TRUE;
         //CmdMessageState.INTERRUPTED : CommandInterrupted := TRUE;
         //CmdMessageState.ABORTED     : CommandAborted     := TRUE;
           CmdMessageState.ERROR       : Error              := TRUE;
				 END_CASE
       
         // Done, Aborted or Error ?
         IF (_response.State >= CmdMessageState.DONE )
         THEN
           // Update results
           //OutCmd.Dummy := _response.Dummy;
           // set timeout
           SetTimeout(PT := _timeoutCmd, rTimer := _timerCmd);
           // inc step counter
          _stepCmd := _stepCmd + 1; 
				 END_IF
       END_IF

  03: Done := TRUE;
  
      IF ( NOT Execute)
      THEN
        // reset step counter
       _stepCmd := 0;
        // reset done flag
        Done := FALSE;
        // reset busy flag
        Busy := FALSE;    
        // reset buffered flag
        CommandBuffered := FALSE;  
			END_IF     
ELSE
  // invalid step
  ErrorID := RobotLibraryEvents.ERR_INVALID_STEP;
END_CASE


// Cancel 
IF (Busy) AND (NOT Execute) 
THEN
  // try to remove cmd
  AxesGroup.Acyclic.ActiveCommandRegister.RemoveCmd(_uniqueID);
END_IF


// Reset FB
IF ( NOT Execute )
THEN
 _uniqueId        := 0;
 _stepCmd         := 0;
  Done            := FALSE;
  Busy            := FALSE;
  CommandBuffered := FALSE;
  Error           := FALSE;
  ErrorID         := 0;
  WarningID       := 0;
  InfoID          := 0;  
END_IF
                      
END_METHOD

METHOD ParseResponsePayload : DINT
VAR_INPUT
  /// Response data
  ResponseData : RecvData;
END_VAR
                        // Table 6-212: Received CMD payload (RC to PLC) of "ActivateWorkArea"
// --------------------------
// Header
// --------------------------
// Byte 00 : USINT - ParSeq | State     
// Byte 01 : SINT  - AlarmMessageSeverity    
// Byte 02 : UINT  - AlarmMessageCode HB
// Byte 03 :       - AlarmMessageCode LB

// call base implementation to parse the header from payload buffer
SUPER^.ParseResponseData(ResponseData);

// copy parsed header to response
_response.ParSeq               := _rspHeader.ParSeq;
_response.State                := _rspHeader.State;
_response.AlarmMessageSeverity := _rspHeader.AlarmMessageSeverity;
_response.AlarmMessageCode     := _rspHeader.AlarmMessageCode;
                      
END_METHOD
END_FUNCTION_BLOCK

/// Cancel currently active move command and continue with the next buffered command
FUNCTION_BLOCK ActivateNextCommandFB EXTENDS RobotLibraryBaseFB
// ------------------------------------------------------------------------- 
//  SRCI Robot Library                                                
// ------------------------------------------------------------------------- 
//                                                                           
//  Object:      ActivateNextCommandFB                                       
//  Author:      Thorsten Brach                                                
//  Date:        2024-06-01
//
//  Description:                                              
//   
//                                                                           
//  Copyright: 
//    (C) 2024 Thorsten Brach. All rights reserved                                                                         
//                                                                           
//  Disclaimer:                                                                           
//    This project is provided without any guarantee and can be used for   
//    private and commercial purposes. Any commercial use is at the user’s 
//    own risk and responsibility.
//
// -------------------------------------------------------------------------
VAR_INPUT
  /// Start of the command at the rising edge
  Execute         : BOOL;
  /// Command parameter 
  ParCmd          : ActivateNextCommandParCmd;
END_VAR
VAR_OUTPUT
  /// The command has been completed successfully
  Done            : BOOL;
  /// FB is being processed
  Busy            : BOOL;
  /// Command is transferred and confirmed by the RC
  CommandBuffered : BOOL;
  /// command results
  OutCmd          : ActivateNextCommandOutCmd;
END_VAR

VAR
  /// internal copy of command parameter 
 _parCmd          : ActivateNextCommandParCmd;
  /// command data to send
 _command         : ActivateNextCommandSendData;
  /// response data received
 _response        : ActivateNextCommandRecvData;   
  /// Trigger related EmitterID
 _emitterID       : ARRAY[0..3] OF SINT;
END_VAR

                  
                

METHOD CheckParameterChanged : BOOL
                        // compare memory 
CheckParameterChanged := ( MemCmp(ADR(ParCmd), ADR(_parCmd), SIZEOF(ParCmd)) = RobotLibraryConstants.OK );

IF ( CheckParameterChanged )
THEN  
  // update internal copy of parameters 
 _parCmd := ParCmd;
  // inc parameter sequence
 _command.ParSeq := _command.ParSeq + 1;
  // update command data  
  CommandData := CreateCommandData(); // ( Access via reference to rCommandFB in ACR )
END_IF
                      
END_METHOD

METHOD CreateCommandData : SendData
                        // Table 6-662: Sent CMD payload (PLC to RC) of "ActivateNextCommand"

// --------------------------
// Header
// --------------------------
// Byte 00 : UINT  - Type HB     
// Byte 01 :       - Type LB    
// Byte 02 : USINT - Reserve | ExecutionMode
// Byte 03 : USINT - ParSeq  | Priority
// --------------------------
// Datablock
// --------------------------
// Byte 04 : SINT - EmitterID[0]
// Byte 05 : SINT - EmitterID[1]
// Byte 06 : SINT - EmitterID[2]   
// Byte 07 : SINT - EmitterID[3]
// Byte 08 : SINT - ListenerID
// Byte 09 : BYTE - Reserve

// --------------------------

// set command parameter 
_command.CmdTyp     :=  CmdType.ActivateNextCommand;
_command.ExecMode   :=  ExecutionMode.PARALLEL;
_command.ParSeq     := _command.ParSeq;
_command.Priority   :=  PriorityLevel.NORMAL;
_command.ListenerID := _parCmd.ListenerID;


// copy command data to header
_cmdHeader := _command;
// call base implementation to copy header to payload buffer
SUPER^.CreateCommandData();

// add command.EmitterID[0]
CreateCommandData.AddSint(_command.EmitterID[0]);
// add command.EmitterID[1]
CreateCommandData.AddSint(_command.EmitterID[1]);
// add command.EmitterID[2]
CreateCommandData.AddSint(_command.EmitterID[2]);
// add command.EmitterID[3]
CreateCommandData.AddSint(_command.EmitterID[3]);
// add command.ListenerID
CreateCommandData.AddSint(_command.ListenerID);
// add command.Reserve
CreateCommandData.AddByte(_command.Reserve);
                      
END_METHOD

METHOD PROTECTED OnCall
VAR_IN_OUT
  /// Robot assignment of function
  AxesGroup : AxesGroup; 
END_VAR
                        CASE _stepCmd OF
  
  00:  IF ( Execute ) 
       THEN
         // set busy flag
         Busy := TRUE;
         // Reset command outputs
         MemSet(ADR(OutCmd),0,SIZEOF(OutCmd));
         // apply command parameter
        _parCmd := ParCmd;
         // init parameter sequence
        _command.ParSeq := 1;
         // set timeout
         SetTimeout(PT := _timeoutCmd, rTimer := _timerCmd);
         // inc step counter
        _stepCmd := _stepCmd + 1; 
	     END_IF
     
  01:  // create command data
       CommandData := CreateCommandData();
       // Add command to active command register
      _uniqueID := AxesGroup.Acyclic.ActiveCommandRegister.AddCmd( rCommandFB := THIS^ );     
       // set timeout
       SetTimeout(PT := _timeoutCmd, rTimer := _timerCmd);
       // inc step counter
      _stepCmd := _stepCmd + 1; 

  02:  // Wait for responce received
       IF ( _responseReceived )
       THEN
         // reset response received flag
        _responseReceived := FALSE;

         CASE  _response.State 
         OF
           CmdMessageState.BUFFERED    : CommandBuffered    := TRUE;
         //CmdMessageState.ACTIVE      : Active             := TRUE;
         //CmdMessageState.INTERRUPTED : CommandInterrupted := TRUE;
         //CmdMessageState.ABORTED     : CommandAborted     := TRUE;
           CmdMessageState.ERROR       : Error              := TRUE;
				 END_CASE

         // Done, Aborted or Error ?
         IF (_response.State >= CmdMessageState.DONE )
         THEN
           // Update results
           OutCmd.InvocationCounter := _response.InvocationCounter;
           OutCmd.OriginID          := _response.OriginID;
           // set timeout
           SetTimeout(PT := _timeoutCmd, rTimer := _timerCmd);
           // inc step counter
          _stepCmd := _stepCmd + 1; 
				 END_IF
       END_IF

  03: Done := TRUE;
  
      IF ( NOT Execute)
      THEN
        // reset step counter
       _stepCmd := 0;
        // reset done flag
        Done := FALSE;
        // reset busy flag
        Busy := FALSE;    
        // reset buffered flag
        CommandBuffered := FALSE;  
			END_IF     
ELSE
  // invalid step
  ErrorID := RobotLibraryEvents.ERR_INVALID_STEP;
END_CASE


// Cancel 
IF (Busy) AND (NOT Execute) 
THEN
  // try to remove cmd
  AxesGroup.Acyclic.ActiveCommandRegister.RemoveCmd(_uniqueID);
END_IF


// Reset FB
IF ( NOT Execute )
THEN
 _uniqueId        := 0;
 _stepCmd         := 0;
  Done            := FALSE;
  Busy            := FALSE;
  CommandBuffered := FALSE;
  Error           := FALSE;
  ErrorID         := 0;
  WarningID       := 0;
  InfoID          := 0;  
END_IF
                      
END_METHOD

METHOD ParseResponsePayload : DINT
VAR_INPUT
  /// Response data
  ResponseData : RecvData;
END_VAR
                        // Table 6-26: Received CMD payload (RC to PLC) of "EnableRobot"
// --------------------------
// Header
// --------------------------
// Byte 00 : USINT - ParSeq | State     
// Byte 01 : SINT  - AlarmMessageSeverity    
// Byte 02 : UINT  - AlarmMessageCode HB
// Byte 03 :       - AlarmMessageCode LB
// --------------------------
// Datablock
// --------------------------
// Byte 04 : USINT - InvocationCounter
// Byte 05 : SINT  - Reserved
// Byte 06 : INT   - OriginID HB
// Byte 07 : INT   - OriginID LB
// --------------------------

// call base implementation to parse the header from payload buffer
SUPER^.ParseResponseData(ResponseData);

// copy parsed header to response
_response.ParSeq               := _rspHeader.ParSeq;
_response.State                := _rspHeader.State;
_response.AlarmMessageSeverity := _rspHeader.AlarmMessageSeverity;
_response.AlarmMessageCode     := _rspHeader.AlarmMessageCode;

// Get InvocationCounter
_response.InvocationCounter    := ResponseData.GetUsint();
// Get Reserve
_response.Reserve              := ResponseData.GetSint();
// Get OriginID
_response.OriginID             := ResponseData.GetInt();
                      
END_METHOD
END_FUNCTION_BLOCK

/// Activate robot cycle brake test and give feedback to PLC
FUNCTION_BLOCK BrakeTestFB EXTENDS RobotLibraryBaseFB
// ------------------------------------------------------------------------- 
//  SRCI Robot Library                                                
// ------------------------------------------------------------------------- 
//                                                                           
//  Object:      BrakeTest                                       
//  Author:      Thorsten Brach                                                
//  Date:        2024-06-01
//
//  Description:                                              
//   
//                                                                           
//  Copyright: 
//    (C) 2024 Thorsten Brach. All rights reserved                                                                         
//                                                                           
//  Disclaimer:                                                                           
//    This project is provided without any guarantee and can be used for   
//    private and commercial purposes. Any commercial use is at the user’s 
//    own risk and responsibility.
//
// -------------------------------------------------------------------------
VAR_INPUT
  /// Start of the command at the rising edge
  Execute            : BOOL;
  /// Command parameter 
  ParCmd             : BrakeTestParCmd;
END_VAR
VAR_OUTPUT
  /// The command has been completed successfully
  Done               : BOOL;
  /// FB is being processed
  Busy               : BOOL;
  /// Command is transferred and confirmed by the RC
  CommandBuffered    : BOOL;
  /// During the realization of the brake test, the command controls the motion of the respective axis group.
  /// TRUE: The brake test is being realized
  /// FALSE: The brake test is not realized
  Active             : BOOL;
  /// The command was aborted by another command.
  CommandAborted     : BOOL;
  /// TRUE, while command is interrupted during execution and can be continued
  CommandInterrupted : BOOL; 
  /// Command output 
  OutCmd             : BrakeTestOutCmd;
END_VAR

var
  /// internal copy of command parameter 
 _parCmd             : BrakeTestParCmd;
  /// command data to send
 _command            : BrakeTestSendData;
  /// response data received
 _response           : BrakeTestRecvData;      
END_VAR

                  
                

METHOD CheckParameterChanged : BOOL
                        // compare memory 
CheckParameterChanged := ( MemCmp(ADR(ParCmd), ADR(_parCmd), SIZEOF(ParCmd)) = RobotLibraryConstants.OK );

IF ( CheckParameterChanged )
THEN  
  // update internal copy of parameters 
 _parCmd := ParCmd;
  // inc parameter sequence
 _command.ParSeq := _command.ParSeq + 1;
  // update command data  
  CommandData := CreateCommandData(); // ( Access via reference to rCommandFB in ACR )
END_IF
                      
END_METHOD

METHOD CreateCommandData : SendData
                        // Table 6-740: Sent CMD payload (PLC to RC) of "BrakeTest"

// --------------------------
// Header
// --------------------------
// Byte 00 : UINT  - Type HB     
// Byte 01 :       - Type LB    
// Byte 02 : USINT - Reserve | ExecutionMode
// Byte 03 : USINT - ParSeq  | Priority
// --------------------------
// Datablock
// --------------------------
// Byte 04 : BYTE - RobotAxesActive
// Byte 05 : BYTE - ExternalAxesActive
// --------------------------

// set command parameter 
_command.CmdTyp               :=  CmdType.BrakeTest;
_command.ExecMode             :=  ExecutionMode.PARALLEL;
_command.ParSeq               := _command.ParSeq;
_command.Priority             :=  PriorityLevel.NORMAL;
_command.RobotAxesActive.0    := _parCmd.RobotAxesActive.Bit00;
_command.RobotAxesActive.1    := _parCmd.RobotAxesActive.AxisJ1;
_command.RobotAxesActive.2    := _parCmd.RobotAxesActive.AxisJ2;
_command.RobotAxesActive.3    := _parCmd.RobotAxesActive.AxisJ3;
_command.RobotAxesActive.4    := _parCmd.RobotAxesActive.AxisJ4;
_command.RobotAxesActive.5    := _parCmd.RobotAxesActive.AxisJ5;
_command.RobotAxesActive.6    := _parCmd.RobotAxesActive.AxisJ6;
_command.RobotAxesActive.7    := _parCmd.RobotAxesActive.Bit07;
_command.ExternalAxesActive.0 := _parCmd.ExternalAxesActive.Bit00;
_command.ExternalAxesActive.1 := _parCmd.ExternalAxesActive.AxisE1;
_command.ExternalAxesActive.2 := _parCmd.ExternalAxesActive.AxisE2;
_command.ExternalAxesActive.3 := _parCmd.ExternalAxesActive.AxisE3;
_command.ExternalAxesActive.4 := _parCmd.ExternalAxesActive.AxisE4;
_command.ExternalAxesActive.5 := _parCmd.ExternalAxesActive.AxisE5;
_command.ExternalAxesActive.6 := _parCmd.ExternalAxesActive.AxisE6;
_command.ExternalAxesActive.7 := _parCmd.ExternalAxesActive.Bit07;

// copy command data to header
_cmdHeader := _command;
// call base implementation to copy header to payload buffer
SUPER^.CreateCommandData();

// add command.EmitterID[0]
CreateCommandData.AddByte(_command.RobotAxesActive);
// add command.EmitterID[1]
CreateCommandData.AddByte(_command.ExternalAxesActive);
                      
END_METHOD

METHOD PROTECTED OnCall
VAR_IN_OUT
  /// Robot assignment of function
  AxesGroup : AxesGroup; 
END_VAR
                        CASE _stepCmd OF
  
  00:  IF ( Execute ) 
       THEN
         // set busy flag
         Busy := TRUE;
         // Reset command outputs
         MemSet(ADR(OutCmd),0,SIZEOF(OutCmd));         
         // apply command parameter
        _parCmd := ParCmd;
         // init parameter sequence
        _command.ParSeq := 1;
         // set timeout
         SetTimeout(PT := _timeoutCmd, rTimer := _timerCmd);
         // inc step counter
        _stepCmd := _stepCmd + 1; 
	     END_IF
     
  01:  // create command data
       CommandData := CreateCommandData();
       // Add command to active command register
      _uniqueID := AxesGroup.Acyclic.ActiveCommandRegister.AddCmd( rCommandFB := THIS^ );     
       // set timeout
       SetTimeout(PT := _timeoutCmd, rTimer := _timerCmd);
       // inc step counter
      _stepCmd := _stepCmd + 1; 

  02:  // Wait for responce received
       IF ( _responseReceived )
       THEN
         // reset response received flag
        _responseReceived := FALSE;

         CASE  _response.State 
         OF
           CmdMessageState.BUFFERED    : CommandBuffered    := TRUE;
           CmdMessageState.ACTIVE      : Active             := TRUE;
           CmdMessageState.INTERRUPTED : CommandInterrupted := TRUE;
           CmdMessageState.ABORTED     : CommandAborted     := TRUE;
           CmdMessageState.ERROR       : Error              := TRUE;
				 END_CASE
                
         // Done, Aborted or Error ?
         IF (_response.State >= CmdMessageState.DONE )
         THEN
           // Update results
           OutCmd.RobotAxesStatus.Bit00     := _response.RobotAxesStatus.0;
           OutCmd.RobotAxesStatus.AxisJ1    := _response.RobotAxesStatus.1;
           OutCmd.RobotAxesStatus.AxisJ2    := _response.RobotAxesStatus.2;
           OutCmd.RobotAxesStatus.AxisJ3    := _response.RobotAxesStatus.3;
           OutCmd.RobotAxesStatus.AxisJ4    := _response.RobotAxesStatus.4;
           OutCmd.RobotAxesStatus.AxisJ5    := _response.RobotAxesStatus.5;
           OutCmd.RobotAxesStatus.AxisJ6    := _response.RobotAxesStatus.6;
           OutCmd.RobotAxesStatus.Bit07     := _response.RobotAxesStatus.7;
           
           OutCmd.RobotAxesWarning.Bit00     := _response.RobotAxesWarning.0;
           OutCmd.RobotAxesWarning.AxisJ1    := _response.RobotAxesWarning.1;
           OutCmd.RobotAxesWarning.AxisJ2    := _response.RobotAxesWarning.2;
           OutCmd.RobotAxesWarning.AxisJ3    := _response.RobotAxesWarning.3;
           OutCmd.RobotAxesWarning.AxisJ4    := _response.RobotAxesWarning.4;
           OutCmd.RobotAxesWarning.AxisJ5    := _response.RobotAxesWarning.5;
           OutCmd.RobotAxesWarning.AxisJ6    := _response.RobotAxesWarning.6;
           OutCmd.RobotAxesWarning.Bit07     := _response.RobotAxesWarning.7;

           OutCmd.ExternalAxesStatus.Bit00   := _response.ExternalAxesStatus.0;
           OutCmd.ExternalAxesStatus.AxisE1  := _response.ExternalAxesStatus.1;
           OutCmd.ExternalAxesStatus.AxisE2  := _response.ExternalAxesStatus.2;
           OutCmd.ExternalAxesStatus.AxisE3  := _response.ExternalAxesStatus.3;
           OutCmd.ExternalAxesStatus.AxisE4  := _response.ExternalAxesStatus.4;
           OutCmd.ExternalAxesStatus.AxisE5  := _response.ExternalAxesStatus.5;
           OutCmd.ExternalAxesStatus.AxisE6  := _response.ExternalAxesStatus.6;
           OutCmd.ExternalAxesStatus.Bit07   := _response.ExternalAxesStatus.7;

           OutCmd.ExternalAxesWarning.Bit00  := _response.ExternalAxesWarning.0;
           OutCmd.ExternalAxesWarning.AxisE1 := _response.ExternalAxesWarning.1;
           OutCmd.ExternalAxesWarning.AxisE2 := _response.ExternalAxesWarning.2;
           OutCmd.ExternalAxesWarning.AxisE3 := _response.ExternalAxesWarning.3;
           OutCmd.ExternalAxesWarning.AxisE4 := _response.ExternalAxesWarning.4;
           OutCmd.ExternalAxesWarning.AxisE5 := _response.ExternalAxesWarning.5;
           OutCmd.ExternalAxesWarning.AxisE6 := _response.ExternalAxesWarning.6;
           OutCmd.ExternalAxesWarning.Bit07  := _response.ExternalAxesWarning.7;
           
           // set timeout
           SetTimeout(PT := _timeoutCmd, rTimer := _timerCmd);
           // inc step counter
          _stepCmd := _stepCmd + 1; 
				 END_IF
       END_IF

  03: Done := TRUE;
  
      IF ( NOT Execute)
      THEN
        // reset step counter
       _stepCmd := 0;
        // reset done flag
        Done := FALSE;
        // reset busy flag
        Busy := FALSE;    
        // reset buffered flag
        CommandBuffered := FALSE;  
			END_IF     
ELSE
  // invalid step
  ErrorID := RobotLibraryEvents.ERR_INVALID_STEP;
END_CASE


// Cancel 
IF (Busy) AND (NOT Execute) 
THEN
  // try to remove cmd
  AxesGroup.Acyclic.ActiveCommandRegister.RemoveCmd(_uniqueID);
END_IF


// Reset FB
IF ( NOT Execute )
THEN
 _uniqueId           := 0;
 _stepCmd            := 0;
  Done               := FALSE;
  Busy               := FALSE;
  Active             := FALSE;
  CommandBuffered    := FALSE;
  CommandInterrupted := FALSE;
  CommandAborted     := FALSE;
  Error              := FALSE;
  ErrorID            := 0;
  WarningID          := 0;
  InfoID             := 0;  
END_IF
                      
END_METHOD

METHOD ParseResponsePayload : DINT
VAR_INPUT
  /// Response data
  ResponseData : RecvData;
END_VAR
                        // Table 6-741: Received CMD payload (RC to PLC) of "BrakeTest"
// --------------------------
// Header
// --------------------------
// Byte 00 : USINT - ParSeq | State     
// Byte 01 : SINT  - AlarmMessageSeverity    
// Byte 02 : UINT  - AlarmMessageCode HB
// Byte 03 :       - AlarmMessageCode LB
// --------------------------
// Datablock
// --------------------------
// Byte 04 : BYTE  - RobotAxesStatus
// Byte 05 : BYTE  - ExternalAxesStatus
// Byte 06 : BYTE  - RobotAxesWarning
// Byte 07 : BYTE  - ExternalAxesWarning
// --------------------------

// call base implementation to parse the header from payload buffer
SUPER^.ParseResponseData(ResponseData);

// copy parsed header to response
_response.ParSeq               := _rspHeader.ParSeq;
_response.State                := _rspHeader.State;
_response.AlarmMessageSeverity := _rspHeader.AlarmMessageSeverity;
_response.AlarmMessageCode     := _rspHeader.AlarmMessageCode;

// Get RobotAxesStatus
_response.RobotAxesStatus     := ResponseData.GetByte();
// Get ExternalAxesStatus
_response.ExternalAxesStatus  := ResponseData.GetByte();
// Get RobotAxesWarning
_response.RobotAxesWarning    := ResponseData.GetByte();
// Get ExternalAxesWarning
_response.ExternalAxesWarning := ResponseData.GetByte();
                      
END_METHOD
END_FUNCTION_BLOCK

/// Release robot arm’s brakes.
FUNCTION_BLOCK OpenBrakeFB EXTENDS RobotLibraryBaseFB
// ------------------------------------------------------------------------- 
//  SRCI Robot Library                                                
// ------------------------------------------------------------------------- 
//                                                                           
//  Object:      OpenBrakeFB                                       
//  Author:      Thorsten Brach                                                
//  Date:        2024-06-01
//
//  Description:                                              
//   
//                                                                           
//  Copyright: 
//    (C) 2024 Thorsten Brach. All rights reserved                                                                         
//                                                                           
//  Disclaimer:                                                                           
//    This project is provided without any guarantee and can be used for   
//    private and commercial purposes. Any commercial use is at the user’s 
//    own risk and responsibility.
//
// -------------------------------------------------------------------------
VAR_INPUT
  /// Start of the command at the rising edge
  Execute            : BOOL;
  /// Command parameter 
  ParCmd             : OpenBrakeParCmd;  
END_VAR

VAR_OUTPUT
  /// FB is being processed
  Busy              : BOOL;
  /// Command is transferred and confirmed by the RC
  CommandBuffered   : BOOL;
  /// Receiving of input parameter values has been acknowledged by RC
  ParameterAccepted : BOOL;
  /// Command output 
  OutCmd            : OpenBrakeOutCmd;  
END_VAR

VAR
  /// internal copy of command parameter 
 _parCmd             : OpenBrakeParCmd;
  /// command data to send
 _command            : OpenBrakeSendData;
  /// response data received
 _response           : OpenBrakeRecvData;      
END_VAR

                  
                

METHOD CheckParameterChanged : BOOL
                        // compare memory 
CheckParameterChanged := ( MemCmp(ADR(ParCmd), ADR(_parCmd), SIZEOF(ParCmd)) = RobotLibraryConstants.OK );

IF ( CheckParameterChanged )
THEN  
  // update internal copy of parameters 
 _parCmd := ParCmd;
  // inc parameter sequence
 _command.ParSeq := _command.ParSeq + 1;
  // update command data  
  CommandData := CreateCommandData(); // ( Access via reference to rCommandFB in ACR )
END_IF
                      
END_METHOD

METHOD CreateCommandData : SendData
                        // Table 6-681: Sent CMD payload (PLC to RC) of "OpenBrake"

// --------------------------
// Header
// --------------------------
// Byte 00 : UINT  - Type HB     
// Byte 01 :       - Type LB    
// Byte 02 : USINT - Reserve | ExecutionMode
// Byte 03 : USINT - ParSeq  | Priority
// --------------------------
// Datablock
// --------------------------
// Byte 04 : BYTE - RobotAxesBrakeRelease
// Byte 05 : BYTE - ExternalAxesBrakeRelease
// --------------------------

// set command parameter 
_command.CmdTyp                     :=  CmdType.OpenBrake;
_command.ExecMode                   :=  ExecutionMode.PARALLEL;
_command.ParSeq                     := _command.ParSeq;
_command.Priority                   :=  PriorityLevel.NORMAL;
_command.RobotAxesBrakeRelease.0    := _parCmd.RobotAxesBrakeRelease   .Bit00;
_command.RobotAxesBrakeRelease.1    := _parCmd.RobotAxesBrakeRelease   .AxisJ1;
_command.RobotAxesBrakeRelease.2    := _parCmd.RobotAxesBrakeRelease   .AxisJ2;
_command.RobotAxesBrakeRelease.3    := _parCmd.RobotAxesBrakeRelease   .AxisJ3;
_command.RobotAxesBrakeRelease.4    := _parCmd.RobotAxesBrakeRelease   .AxisJ4;
_command.RobotAxesBrakeRelease.5    := _parCmd.RobotAxesBrakeRelease   .AxisJ5;
_command.RobotAxesBrakeRelease.6    := _parCmd.RobotAxesBrakeRelease   .AxisJ6;
_command.RobotAxesBrakeRelease.7    := _parCmd.RobotAxesBrakeRelease   .Bit07;
_command.ExternalAxesBrakeRelease.0 := _parCmd.ExternalAxesBrakeRelease.Bit00;
_command.ExternalAxesBrakeRelease.1 := _parCmd.ExternalAxesBrakeRelease.AxisE1;
_command.ExternalAxesBrakeRelease.2 := _parCmd.ExternalAxesBrakeRelease.AxisE2;
_command.ExternalAxesBrakeRelease.3 := _parCmd.ExternalAxesBrakeRelease.AxisE3;
_command.ExternalAxesBrakeRelease.4 := _parCmd.ExternalAxesBrakeRelease.AxisE4;
_command.ExternalAxesBrakeRelease.5 := _parCmd.ExternalAxesBrakeRelease.AxisE5;
_command.ExternalAxesBrakeRelease.6 := _parCmd.ExternalAxesBrakeRelease.AxisE6;
_command.ExternalAxesBrakeRelease.7 := _parCmd.ExternalAxesBrakeRelease.Bit07;


// copy command data to header
_cmdHeader := _command;
// call base implementation to copy header to payload buffer
SUPER^.CreateCommandData();

// add command.EmitterID[0]
CreateCommandData.AddByte(_command.RobotAxesBrakeRelease);
// add command.EmitterID[1]
CreateCommandData.AddByte(_command.ExternalAxesBrakeRelease);
                      
END_METHOD

METHOD PROTECTED OnCall
VAR_IN_OUT
  /// Robot assignment of function
  AxesGroup : AxesGroup; 
END_VAR
                        CASE _stepCmd OF
  
  00:  IF ( Execute ) 
       THEN
         // set busy flag
         Busy := TRUE;
         // Reset command outputs
         MemSet(ADR(OutCmd),0,SIZEOF(OutCmd));         
         // apply command parameter
        _parCmd := ParCmd;
         // init parameter sequence
        _command.ParSeq := 1;
         // set timeout
         SetTimeout(PT := _timeoutCmd, rTimer := _timerCmd);
         // inc step counter
        _stepCmd := _stepCmd + 1; 
	     END_IF
     
  01:  // create command data
       CommandData := CreateCommandData();
       // Add command to active command register
      _uniqueID := AxesGroup.Acyclic.ActiveCommandRegister.AddCmd( rCommandFB := THIS^ );     
       // set timeout
       SetTimeout(PT := _timeoutCmd, rTimer := _timerCmd);
       // inc step counter
      _stepCmd := _stepCmd + 1; 

  02:  // Wait for responce received
       IF ( _responseReceived )
       THEN
         // reset response received flag
        _responseReceived := FALSE;

         CASE  _response.State 
         OF
           CmdMessageState.BUFFERED    : CommandBuffered    := TRUE;
           CmdMessageState.ACTIVE      : ParameterAccepted  := TRUE;           
           CmdMessageState.ERROR       : Error              := TRUE;
				 END_CASE
                
         // Done, Aborted or Error ?
         IF (_response.State >= CmdMessageState.DONE )
         THEN
           // Update results
           OutCmd.Enabled                          := _response.Enabled.0;
           OutCmd.RobotAxesBrakeReleased.Bit00     := _response.RobotAxesBrakeReleased.0;
           OutCmd.RobotAxesBrakeReleased.AxisJ1    := _response.RobotAxesBrakeReleased.1;
           OutCmd.RobotAxesBrakeReleased.AxisJ2    := _response.RobotAxesBrakeReleased.2;
           OutCmd.RobotAxesBrakeReleased.AxisJ3    := _response.RobotAxesBrakeReleased.3;
           OutCmd.RobotAxesBrakeReleased.AxisJ4    := _response.RobotAxesBrakeReleased.4;
           OutCmd.RobotAxesBrakeReleased.AxisJ5    := _response.RobotAxesBrakeReleased.5;
           OutCmd.RobotAxesBrakeReleased.AxisJ6    := _response.RobotAxesBrakeReleased.6;
           OutCmd.RobotAxesBrakeReleased.Bit07     := _response.RobotAxesBrakeReleased.7;
           OutCmd.ExternalAxesBrakeReleased.Bit00  := _response.ExternalAxesBrakeReleased.0;
           OutCmd.ExternalAxesBrakeReleased.AxisE1 := _response.ExternalAxesBrakeReleased.1;
           OutCmd.ExternalAxesBrakeReleased.AxisE2 := _response.ExternalAxesBrakeReleased.2;
           OutCmd.ExternalAxesBrakeReleased.AxisE3 := _response.ExternalAxesBrakeReleased.3;
           OutCmd.ExternalAxesBrakeReleased.AxisE4 := _response.ExternalAxesBrakeReleased.4;
           OutCmd.ExternalAxesBrakeReleased.AxisE5 := _response.ExternalAxesBrakeReleased.5;
           OutCmd.ExternalAxesBrakeReleased.AxisE6 := _response.ExternalAxesBrakeReleased.6;
           OutCmd.ExternalAxesBrakeReleased.Bit07  := _response.ExternalAxesBrakeReleased.7;

           // set timeout
           SetTimeout(PT := _timeoutCmd, rTimer := _timerCmd);
           // inc step counter
          _stepCmd := _stepCmd + 1; 
				 END_IF
       END_IF

  03: IF ( NOT Execute)
      THEN
        // reset step counter
       _stepCmd := 0;
        // reset busy flag
        Busy := FALSE;    
        // reset buffered flag
        CommandBuffered := FALSE;  
        // reset parameter accepted flag
        ParameterAccepted := FALSE;
			END_IF     
ELSE
  // invalid step
  ErrorID := RobotLibraryEvents.ERR_INVALID_STEP;
END_CASE


// Cancel 
IF (Busy) AND (NOT Execute) 
THEN
  // try to remove cmd
  AxesGroup.Acyclic.ActiveCommandRegister.RemoveCmd(_uniqueID);
END_IF


// Reset FB
IF ( NOT Execute )
THEN
 _uniqueId           := 0;
 _stepCmd            := 0;
  Busy               := FALSE;
  CommandBuffered    := FALSE;
  ParameterAccepted  := FALSE;
  Error              := FALSE;
  ErrorID            := 0;
  WarningID          := 0;
  InfoID             := 0;  
END_IF
                      
END_METHOD

METHOD ParseResponsePayload : DINT
VAR_INPUT
  /// Response data
  ResponseData : RecvData;
END_VAR
                        // Table 6-741: Received CMD payload (RC to PLC) of "BrakeTest"
// --------------------------
// Header
// --------------------------
// Byte 00 : USINT - ParSeq | State     
// Byte 01 : SINT  - AlarmMessageSeverity    
// Byte 02 : UINT  - AlarmMessageCode HB
// Byte 03 :       - AlarmMessageCode LB
// --------------------------
// Datablock
// --------------------------
// Byte 04 : BOOL  - Enabled
// Byte 05 : BYTE  - RobotAxesBrakeReleased
// Byte 06 : BYTE  - ExternalAxesBrakeReleased
// --------------------------

// call base implementation to parse the header from payload buffer
SUPER^.ParseResponseData(ResponseData);

// copy parsed header to response
_response.ParSeq               := _rspHeader.ParSeq;
_response.State                := _rspHeader.State;
_response.AlarmMessageSeverity := _rspHeader.AlarmMessageSeverity;
_response.AlarmMessageCode     := _rspHeader.AlarmMessageCode;

// Get RobotAxesStatus
_response.RobotAxesBrakeReleased     := ResponseData.GetByte();
// Get ExternalAxesStatus
_response.ExternalAxesBrakeReleased  := ResponseData.GetByte();

                      
END_METHOD
END_FUNCTION_BLOCK

/// Calculate cartesian position from existing cartesian position
FUNCTION_BLOCK CalculateCartesianPositionFB EXTENDS RobotLibraryBaseFB
// ------------------------------------------------------------------------- 
//  SRCI Robot Library                                                
// ------------------------------------------------------------------------- 
//                                                                           
//  Object:      CalculateCartesianPositionFB                                       
//  Author:      Thorsten Brach                                                
//  Date:        2024-06-01
//
//  Description:                                              
//   
//                                                                           
//  Copyright: 
//    (C) 2024 Thorsten Brach. All rights reserved                                                                         
//                                                                           
//  Disclaimer:                                                                           
//    This project is provided without any guarantee and can be used for   
//    private and commercial purposes. Any commercial use is at the user’s 
//    own risk and responsibility.
//
// -------------------------------------------------------------------------
VAR_INPUT
  /// Start of the command at the rising edge
  Execute            : BOOL;
  /// Command parameter 
  ParCmd             : CalculateCartesianPositionParCmd;  
END_VAR

VAR_OUTPUT
  /// The command has been completed successfully
  Done               : BOOL;
  /// FB is being processed
  Busy               : BOOL;
  /// Command is transferred and confirmed by the RC
  CommandBuffered    : BOOL;
  /// Command output 
  OutCmd            : CalculateCartesianPositionOutCmd;  
END_VAR

VAR
  /// internal copy of command parameter 
 _parCmd             : CalculateCartesianPositionParCmd;
  /// command data to send
 _command            : CalculateCartesianPositionSendData;
  /// response data received
 _response           : CalculateCartesianPositionRecvData;      
END_VAR

                  
                

METHOD CheckParameterChanged : BOOL
                        // compare memory 
CheckParameterChanged := ( MemCmp(ADR(ParCmd), ADR(_parCmd), SIZEOF(ParCmd)) = RobotLibraryConstants.OK );

IF ( CheckParameterChanged )
THEN  
  // update internal copy of parameters 
 _parCmd := ParCmd;
  // inc parameter sequence
 _command.ParSeq := _command.ParSeq + 1;
  // update command data  
  CommandData := CreateCommandData(); // ( Access via reference to rCommandFB in ACR )
END_IF
                      
END_METHOD

METHOD CreateCommandData : SendData
                        // Table 6-681: Sent CMD payload (PLC to RC) of "OpenBrake"

// --------------------------
// Header
// --------------------------
// Byte 00 : UINT  - Type HB     
// Byte 01 :       - Type LB    
// Byte 02 : USINT - Reserve | ExecutionMode
// Byte 03 : USINT - ParSeq  | Priority
// --------------------------
// Datablock
// --------------------------
// Byte 04 : BYTE - RobotAxesBrakeRelease
// Byte 05 : BYTE - ExternalAxesBrakeRelease
// --------------------------

// set command parameter 
_command.CmdTyp                     :=  CmdType.CalculateCartesianPosition;
_command.ExecMode                   :=  ExecutionMode.PARALLEL;
_command.ParSeq                     := _command.ParSeq;
_command.Priority                   :=  PriorityLevel.NORMAL;
_command.FrameNo                    := _parCmd.FrameNo;
_command.TargetFrameNo              := _parCmd.TargetFrameNo;
_command.CartesianPosition          := _parCmd.CartesianPosition;

// copy command data to header
_cmdHeader := _command;
// call base implementation to copy header to payload buffer
SUPER^.CreateCommandData();

// add command.FrameNo
CreateCommandData.AddUsint(_command.FrameNo);
// add command.TargetFrameNo
CreateCommandData.AddUsint(_command.TargetFrameNo);
// add command.CartesianPosition.X
CreateCommandData.AddReal(_command.CartesianPosition.X);
// add command.CartesianPosition.Y
CreateCommandData.AddReal(_command.CartesianPosition.Y);
// add command.CartesianPosition.Z
CreateCommandData.AddReal(_command.CartesianPosition.Z);
// add command.CartesianPosition.Rx
CreateCommandData.AddReal(_command.CartesianPosition.Rx);
// add command.CartesianPosition.Ry
CreateCommandData.AddReal(_command.CartesianPosition.Ry);
// add command.CartesianPosition.Rz
CreateCommandData.AddReal(_command.CartesianPosition.Rz);
// add command.CartesianPosition.Config
CreateCommandData.AddArmConfig(_command.CartesianPosition.Config);
// add command.CartesianPosition.TurnNumber
CreateCommandData.AddTurnNumber(_command.CartesianPosition.TurnNumber);
// add command.CartesianPosition.E1
CreateCommandData.AddReal(_command.CartesianPosition.E1);
// add command.CartesianPosition.E2
CreateCommandData.AddReal(_command.CartesianPosition.E2);
// add command.CartesianPosition.E3
CreateCommandData.AddReal(_command.CartesianPosition.E3);
// add command.CartesianPosition.E4
CreateCommandData.AddReal(_command.CartesianPosition.E4);
// add command.CartesianPosition.E5
CreateCommandData.AddReal(_command.CartesianPosition.E5);
// add command.CartesianPosition.E6
CreateCommandData.AddReal(_command.CartesianPosition.E6);
                      
END_METHOD

METHOD PROTECTED OnCall
VAR_IN_OUT
  /// Robot assignment of function
  AxesGroup : AxesGroup; 
END_VAR
                        CASE _stepCmd OF
  
  00:  IF ( Execute ) 
       THEN
         // set busy flag
         Busy := TRUE;
         // Reset command outputs
         MemSet(ADR(OutCmd),0,SIZEOF(OutCmd));         
         // apply command parameter
        _parCmd := ParCmd;
         // init parameter sequence
        _command.ParSeq := 1;
         // set timeout
         SetTimeout(PT := _timeoutCmd, rTimer := _timerCmd);
         // inc step counter
        _stepCmd := _stepCmd + 1; 
	     END_IF
     
  01:  // create command data
       CommandData := CreateCommandData();
       // Add command to active command register
      _uniqueID := AxesGroup.Acyclic.ActiveCommandRegister.AddCmd( rCommandFB := THIS^ );     
       // set timeout
       SetTimeout(PT := _timeoutCmd, rTimer := _timerCmd);
       // inc step counter
      _stepCmd := _stepCmd + 1; 

  02:  // Wait for responce received
       IF ( _responseReceived )
       THEN
         // reset response received flag
        _responseReceived := FALSE;

         CASE  _response.State 
         OF
           CmdMessageState.BUFFERED    : CommandBuffered    := TRUE;
           CmdMessageState.ERROR       : Error              := TRUE;
				 END_CASE
                
         // Done, Aborted or Error ?
         IF (_response.State >= CmdMessageState.DONE )
         THEN
           // Update results
           OutCmd.TargetToolNoReturn      := _response.TargetToolNoReturn;
           OutCmd.TargetFrameNoReturn     := _response.TargetFrameNoReturn;
           OutCmd.CartesianPositionReturn := _response.CartesianPositionReturn;

           // set timeout
           SetTimeout(PT := _timeoutCmd, rTimer := _timerCmd);
           // inc step counter
          _stepCmd := _stepCmd + 1; 
				 END_IF
       END_IF

  03: Done := TRUE;
      IF ( NOT Execute)
      THEN
        // reset step counter
       _stepCmd := 0;
        // reset done flag
        Done := FALSE;
        // reset busy flag
        Busy := FALSE; 
        // reset buffered flag
        CommandBuffered := FALSE;  
			END_IF     
ELSE
  // invalid step
  ErrorID := RobotLibraryEvents.ERR_INVALID_STEP;
END_CASE


// Cancel 
IF (Busy) AND (NOT Execute) 
THEN
  // try to remove cmd
  AxesGroup.Acyclic.ActiveCommandRegister.RemoveCmd(_uniqueID);
END_IF


// Reset FB
IF ( NOT Execute )
THEN
 _uniqueId           := 0;
 _stepCmd            := 0;
  Done               := FALSE;
  Busy               := FALSE;
  CommandBuffered    := FALSE;
  Error              := FALSE;
  ErrorID            := 0;
  WarningID          := 0;
  InfoID             := 0;  
END_IF
                      
END_METHOD

METHOD ParseResponsePayload : DINT
VAR_INPUT
  /// Response data
  ResponseData : RecvData;
END_VAR
                        // Table 6-741: Received CMD payload (RC to PLC) of "BrakeTest"
// --------------------------
// Header
// --------------------------
// Byte 00 : USINT - ParSeq | State     
// Byte 01 : SINT  - AlarmMessageSeverity    
// Byte 02 : UINT  - AlarmMessageCode HB
// Byte 03 :       - AlarmMessageCode LB
// --------------------------
// Datablock
// --------------------------
// Byte 04 : BOOL  - Enabled
// Byte 05 : BYTE  - RobotAxesBrakeReleased
// Byte 06 : BYTE  - ExternalAxesBrakeReleased
// --------------------------

// call base implementation to parse the header from payload buffer
SUPER^.ParseResponseData(ResponseData);

// copy parsed header to response
_response.ParSeq               := _rspHeader.ParSeq;
_response.State                := _rspHeader.State;
_response.AlarmMessageSeverity := _rspHeader.AlarmMessageSeverity;
_response.AlarmMessageCode     := _rspHeader.AlarmMessageCode;

// Get TargetToolNoReturn
_response.TargetToolNoReturn   := ResponseData.GetUsint();
// Get TargetFrameNoReturn
_response.TargetFrameNoReturn  := ResponseData.GetUsint();
// Get CartesianPositionReturn.X
_response.CartesianPositionReturn.X := ResponseData.GetReal();
// Get CartesianPositionReturn.Y
_response.CartesianPositionReturn.Y := ResponseData.GetReal();
// Get CartesianPositionReturn.Z
_response.CartesianPositionReturn.Z := ResponseData.GetReal();
// Get CartesianPositionReturn.Rx
_response.CartesianPositionReturn.Rx := ResponseData.GetReal();
// Get CartesianPositionReturn.Ry
_response.CartesianPositionReturn.Ry := ResponseData.GetReal();
// Get CartesianPositionReturn.Rz
_response.CartesianPositionReturn.Rz := ResponseData.GetReal();
// Get CartesianPositionReturn.Config
_response.CartesianPositionReturn.Config := ResponseData.GetArmConfig();
// Get CartesianPositionReturn.TurnNumber
_response.CartesianPositionReturn.TurnNumber := ResponseData.GetTurnNumbers();
// Get CartesianPositionReturn.E1
_response.CartesianPositionReturn.E1 := ResponseData.GetReal();
// Get CartesianPositionReturn.E2
_response.CartesianPositionReturn.E2 := ResponseData.GetReal();
// Get CartesianPositionReturn.E3
_response.CartesianPositionReturn.E3 := ResponseData.GetReal();
// Get CartesianPositionReturn.E4
_response.CartesianPositionReturn.E4 := ResponseData.GetReal();
// Get CartesianPositionReturn.E5
_response.CartesianPositionReturn.E5 := ResponseData.GetReal();
// Get CartesianPositionReturn.E6
_response.CartesianPositionReturn.E6 := ResponseData.GetReal();

                      
END_METHOD
END_FUNCTION_BLOCK

